TYPE EspSystemInfo :
STRUCT
	UptimeUs			: ULINT;
	ParentUid			: ULINT;
	HopCount			: BYTE;
	ChildCount			: BYTE;
	StatusFlags			: BYTE;
	Reserved			: BYTE;
	ReportedIp			: T_IPv4Addr;
END_STRUCT
END_TYPE

(* stored: Version 1.1.0.1
   DUT EspSystemInfo: Id {4e920ebd-15f1-4fb6-9c8f-cdfc3bfe0802} *)
